RoboDK station: Coursework2_robot_manipulation.rdk

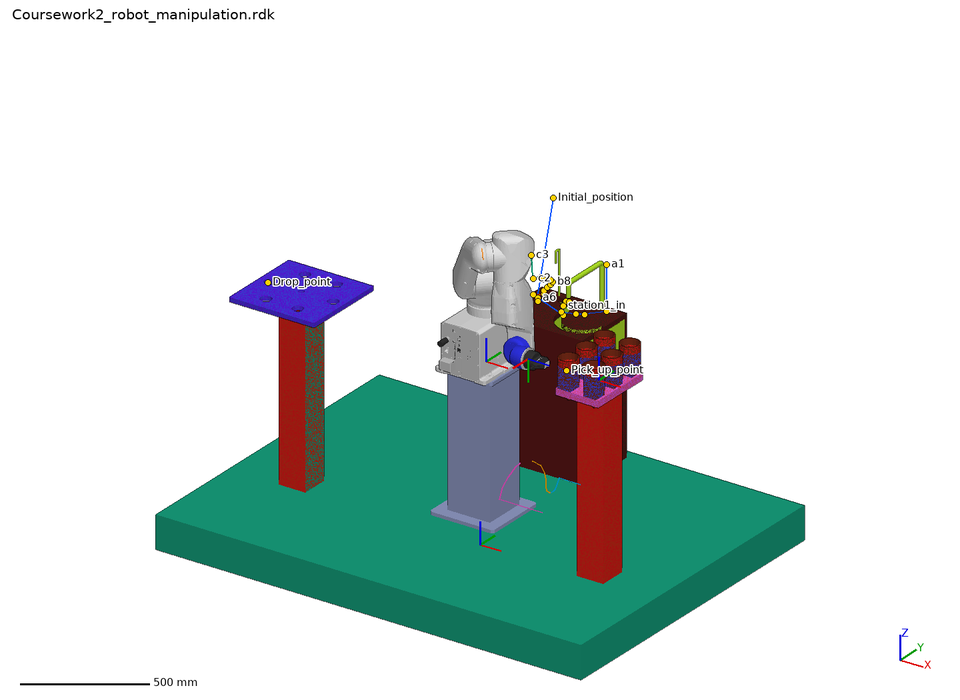
[picture v0: the station drawn from its stored meshes, robots at their saved joint values, targets as dots, program paths as lines]
Station Coursework2_robot_manipulator (saved by RoboDK 5.8.0). Poses are relative to the parent item; angles as X-Y-Z fixed-axis rotations.
Station parameters (name, value as stored): IO_5, 1
  - frame baseframe at (0, 0, 0) mm
    - object PDE4431_CW2_2024 at (0, 0, 0) mm, rotated rx 90 ry 0 rz 0 deg, size 2000 x 980 x 1500 mm, geometry from PDE4431_CW2_2024.STEP
    - frame Epson VT6 Base at (15, 20, 780) mm
      - robot Epson VT6: 6 axes, payload 6 kg, reach 920 mm, repeatability 0.1 mm, weight 40 kg
          modified DH rows (alpha deg, a mm, theta deg, d mm): 0, 0, 0, 412; -90, 100, -90, 0; 0, 420, 0, 0; -90, 0, 0, 400; 90, 0, 0, 0; -90, 0, 0, 80
          base shift (0, 0, 0) mm, rotated rx 0 ry 0 rz 90 deg
          joint limits [-170, -160, -51, -200, -125, -360] to [170, 65, 190, 200, 125, 360]; home [0, 0, 0, 0, 0, 0]; saved at [-133.764, -52.802, -29.005, -135.943, -84.093, 84.313]
        - tool Tool 1, TCP at (0, 0, 180) mm, rotated rx -90 ry 0 rz 0 deg
        - frame RobotiQ 2F-140 Gripper (Mechanism) Base at (0, 0, 0) mm
          - robot RobotiQ 2F-140 Gripper (Mechanism) (model RobotiQ 2F140): 1 axes, payload 5 kg
              joint limits [0] to [140]; home [140]; saved at [60]
    - frame input_area_reference_frame at (700, -200, 980) mm
      - object Cone-Part at (60, -120, 50) mm, rotated rx 90 ry 0 rz 90 deg, size 84.9 x 182 x 85 mm, geometry from Cone-Part.STEP
      - object Cone-Part at (60, 0, 50) mm, rotated rx 90 ry 0 rz 90 deg, size 84.9 x 182 x 85 mm, geometry from Cone-Part.STEP
      - object Cone-Part at (60, 120, 50) mm, rotated rx 90 ry 0 rz 90 deg, size 84.9 x 182 x 85 mm, geometry from Cone-Part.STEP
      - object Cone-Part at (-60, -120, 50) mm, rotated rx 90 ry 0 rz 90 deg, size 84.9 x 182 x 85 mm, geometry from Cone-Part.STEP
      - object Cone-Part at (-60, 0, 50) mm, rotated rx 90 ry 0 rz 90 deg, size 84.9 x 182 x 85 mm, geometry from Cone-Part.STEP
      - object Cone-Part at (-60, 120, 50) mm, rotated rx 90 ry 0 rz 90 deg, size 84.9 x 182 x 85 mm, geometry from Cone-Part.STEP
    - target Initial_position (Cartesian target) at (0, 493.22, 1288.03) mm, rotated rx 138 ry 0 rz 0 deg; joints [3.066, 29.719, -43.422, 4.791, -28.422, -96.269] of Epson VT6
    - target Gripper_open (Cartesian target) at (0.67, 380.04, 1461.97) mm, rotated rx -90 ry 0 rz 0 deg; joints [90, -0.57, 0.57, -89.99, -12.6, 0] of RobotiQ 2F-140 Gripper (Mechanism)
    - target Gripper_closed (Cartesian target) at (0.67, 380.04, 1461.97) mm, rotated rx -90 ry 0 rz 0 deg; joints [60, -0.57, 0.57, -89.99, -12.6, 0] of RobotiQ 2F-140 Gripper (Mechanism)
    - target Pick_up_point (Cartesian target) at (630, -320, 1050) mm, rotated rx 180 ry 0 rz -90 deg; joints [-121.329, -52.273, -41.785, -148.607, -93.465, 92.112] of Epson VT6
    - target station1_in (Cartesian target) at (107.17, 405.57, 892) mm, rotated rx 134.1 ry 22.52 rz 29.53 deg; joints [-42.76, -50.507, -48.896, -94.494, -48.491, -288.218] of Epson VT6
    - target station_in2 (Cartesian target) at (107.17, 425.58, 902) mm, rotated rx 154.09 ry 0 rz 49.53 deg; joints [-46.784, -59.524, -43.679, -90.222, -63.389, -255.291] of Epson VT6
    - target Station1_vert (Cartesian target) at (107.17, 445.58, 892) mm, rotated rx 180 ry 0 rz 49.53 deg; joints [-48.469, -79.022, -29.182, -82.396, -87.508, -251.961] of Epson VT6
    - target station1_return (Cartesian target) at (107.17, 405.57, 892) mm, rotated rx 134.1 ry 22.52 rz 29.53 deg; joints [-42.76, -50.507, -48.896, -94.494, -48.491, -288.218] of Epson VT6
    - target station1_retract2 (Cartesian target) at (107.17, 405.58, 852) mm, rotated rx 134.1 ry 22.52 rz 29.53 deg; joints [-42.76, -58.404, -45.922, -98.782, -49.061, -281.715] of Epson VT6
    - object Pedestal_4 at (14, 3, 150) mm, rotated rx 90 ry 0 rz 0 deg, size 300 x 630 x 300 mm, geometry from Pedestal_4.STEP
    - target Drop_point (Cartesian target) at (-765, -330, 1042) mm, rotated rx 180 ry 0 rz 90 deg; joints [124.2, -59.111, -6.959, -36.632, 70.399, -75.994] of Epson VT6
    - target a1 (Cartesian target) at (249.09, 493.26, 1072) mm, rotated rx 130 ry 0 rz 60.05 deg; joints [-44.186, -25.316, -23.381, -44.941, -61.89, 43.503] of Epson VT6
    - target a2 (Cartesian target) at (249.09, 493.26, 872) mm, rotated rx 130 ry 0 rz 60.05 deg; joints [-44.186, -51.38, -21.842, -59.131, -46.543, 67.327] of Epson VT6
    - target a3 (Cartesian target) at (194.9, 423.42, 872) mm, rotated rx 131.48 ry 11.84 rz 38.12 deg; joints [-47.351, -49.904, -38.58, -79.862, -43.086, 70.249] of Epson VT6
    - target a4 (Cartesian target) at (165.75, 406.79, 872) mm, rotated rx 134.36 ry 21.78 rz 37.08 deg; joints [-48.063, -53.054, -38.624, -75.536, -47.962, 62.433] of Epson VT6
    - target a5 (Cartesian target) at (109.56, 390.77, 872) mm, rotated rx 137.61 ry 29.5 rz 37.51 deg; joints [-45.93, -57.2, -41.919, -79.045, -51.807, 63.625] of Epson VT6
    - target a6 (Cartesian target) at (-2.03, 390.64, 902) mm, rotated rx 167.61 ry 29.5 rz 37.51 deg; joints [-40.605, -82.89, -49.926, -101.486, -85.95, 102.604] of Epson VT6
    - target b1 (Cartesian target) at (-13.32, 409.82, 877) mm, rotated rx 127 ry -33.83 rz -43.76 deg; joints [31.665, -52.224, -39.614, 69.659, -47.778, -224.233] of Epson VT6
    - target b2 (Cartesian target) at (-61.47, 446.95, 877) mm, rotated rx 120 ry 0 rz -61.45 deg; joints [27.592, -42.587, -43.484, 84.177, -30.167, -262.163] of Epson VT6
    - target b3 (Cartesian target) at (-30.23, 471.24, 877) mm, rotated rx 120 ry 0 rz -66.5 deg; joints [22.379, -42.928, -40.487, 79.841, -30.522, -256.952] of Epson VT6
    - target b4 (Cartesian target) at (-44.93, 495.72, 877) mm, rotated rx 120 ry 0 rz -75.12 deg; joints [22.759, -44.277, -33.238, 62.836, -33.826, -247.376] of Epson VT6
    - target b6 (Cartesian target) at (-53.08, 528.17, 877) mm, rotated rx 120 ry 0 rz -85.53 deg; joints [21.649, -46.651, -24.32, 48.543, -39.597, -240.743] of Epson VT6
    - target b7 (Cartesian target) at (-54.53, 553.97, 877) mm, rotated rx 120 ry 0 rz -103.24 deg; joints [19.178, -50.022, -14.03, 34.25, -48.589, -240.495] of Epson VT6
    - target b8 (Cartesian target) at (-65.31, 579.52, 877) mm, rotated rx 120 ry 0 rz -35.21 deg; joints [18.907, -44.258, -33.32, 103.859, -24.661, -245.312] of Epson VT6
    - target b9 (Cartesian target) at (-81.16, 591.33, 877) mm, rotated rx 120 ry 0 rz -15.6 deg; joints [16.379, -43.789, -35.498, 133.999, -21.601, -254.488] of Epson VT6
    - target b10 (Cartesian target) at (-105.52, 575.28, 877) mm, rotated rx 120 ry 0 rz -5.76 deg; joints [17.409, -43.261, -38.323, 149.049, -22.485, -261.342] of Epson VT6
    - target c1 (Cartesian target) at (-126.7, 587.41, 877) mm, rotated rx 121.57 ry -17.23 rz 40.16 deg; joints [13.883, -45.369, -39.632, 180.61, -30.533, -239.449] of Epson VT6
    - target c2 (Cartesian target) at (-143.48, 560.98, 877) mm, rotated rx 121.57 ry -17.23 rz 52.76 deg; joints [12.465, -9.414, 61.191, 171.217, 106.936, -230.002] of Epson VT6
    - target c3 (Cartesian target) at (-146.17, 555.68, 977) mm, rotated rx 127 ry -33.83 rz 40.31 deg; joints [23.435, -32.385, -50.82, 158.038, -42.083, -218.54] of Epson VT6
  - Python program Full1_program (listed below)
  - program Gripper_Open (2 instructions, listed below)
  - program Gripper_close (1 instructions, listed below)
  - program Gripper_fn_detach (1 instructions, listed below)
  - program Gripper_fn_attach (1 instructions, listed below)
  - program Arc1 (15 instructions, listed below)
  - Python program arc1_repeat (listed below)
  - program Arc2 (12 instructions, listed below)
  - Python program arc2_repeat (listed below)
  - program Arc3 (5 instructions, listed below)
  - program Reset_prog (1 instructions, listed below)
  - object Curve1 at (0, 0, 832) mm, geometry from Imported curve
  - machining project Path1 settings: rotZ(0) | rotX(0)*rotY(0) | onStart | onPathStart | onApproach | onPoint | onRetract | onFinish | SetRPM(%1) | SetTool(%1) | Extruder(%1) | default | default | OutOnMov(%1) | OutOffMov(%1) | onPathFinish | M_RunCode(%1)
  - program Path1 (17 instructions, listed below)
  - object Curve2 at (0, 0, 832) mm, geometry from 000000
  - machining project Path2 settings: rotZ(0) | rotX(0)*rotY(0) | onStart | onPathStart | onApproach | onPoint | onRetract | onFinish | SetRPM(%1) | SetTool(%1) | Extruder(%1) | default | default | OutOnMov(%1) | OutOffMov(%1) | onPathFinish | M_RunCode(%1)
  - program Path2 (24 instructions, listed below)
  - object Curve3 at (0, 0, 832) mm
  - machining project Path3 settings: rotZ(0) | rotX(0)*rotY(0) | onStart | onPathStart | onApproach | onPoint | onRetract | onFinish | SetRPM(%1) | SetTool(%1) | Extruder(%1) | default | default | OutOnMov(%1) | OutOffMov(%1) | onPathFinish | M_RunCode(%1)
  - program Path3 (17 instructions, listed below)
  - Python program pick (listed below)
  - Python program drop (listed below)
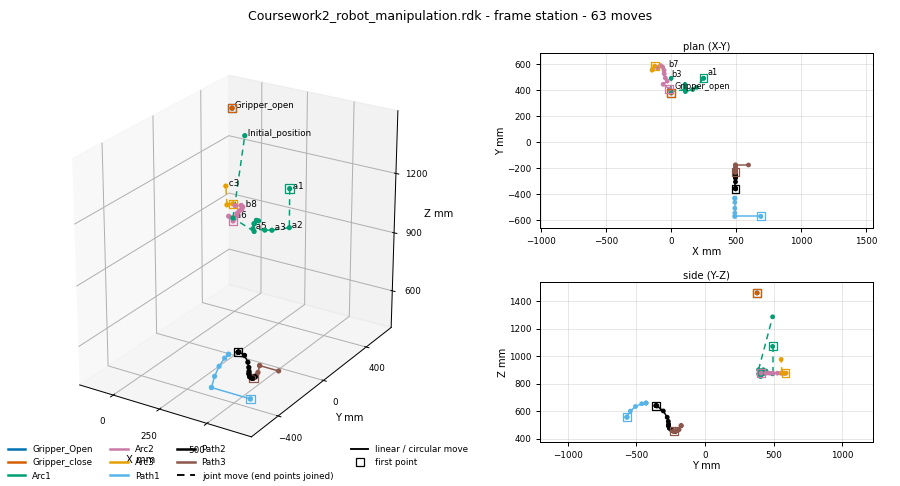
[picture p0: tool path of Coursework2_robot_manipulation.rdk in frame station, 63 of 63 moves have a stored position in this frame; points joined in program order, loops and branches not executed]

--- Python program Full1_program ---
from robodk.robolink import *
from robodk.robomath import *
import time

#Connection b/w roboDK
RDK=Robolink()

#conf. robot
robot=RDK.Item('Epson VT6')

robot.setSpeed(100)

base = RDK.Item('baseframe')
end_effector =RDK.Item('RobotiQ 2F-140 Gripper (Mechanism) Base')

#setting home position
home = RDK.Item('Initial_position')

#Pick_up_points with one point reference
pickup1=RDK.Item('Pick_up_point')
pickup2=pickup1.Pose()*transl(-120,0,0)
pickup3=pickup1.Pose()*transl(-240,0,0)
pickup4=pickup1.Pose()*transl(0,-120,0)
pickup5=pickup1.Pose()*transl(-120,-120,0)
pickup6=pickup1.Pose()*transl(-240,-120,0)

pickup=[pickup3,pickup2,pickup1,pickup6,pickup5,pickup4]

#pickup_approach
pa1=pickup1.Pose()*transl(0,0,-80)
pa2=pickup1.Pose()*transl(-120,0,-80)
pa3=pickup1.Pose()*transl(-240,0,-80)
pa4=pickup1.Pose()*transl(0,-120,-80)
pa5=pickup1.Pose()*transl(-120,-120,-80)
pa6=pickup1.Pose()*transl(-240,-120,-80)

pa7=pickup1.Pose()*transl(-300,-20,-80)

pa=[pa3,pa2,pa1,pa6,pa5,pa4]

#Drop_points with one point reference
drop1=RDK.Item('Drop_point')
drop2=drop1.Pose()*transl(129.9,-75,0)
drop3=drop1.Pose()*transl(259.8,0,0)
drop4=drop1.Pose()*transl(0,150,0)
drop5=drop1.Pose()*transl(129.9,225,0)
drop6=drop1.Pose()*transl(259.8,150,0)



drop=[drop1,drop2,drop3,drop4,drop5,drop6]

#drop_approach
da1=drop1.Pose()*transl(0,0,-80)
da2=drop1.Pose()*transl(129.9,-75,-80)
da3=drop1.Pose()*transl(259.8,0,-80)
da4=drop1.Pose()*transl(0,150,-80)
da5=drop1.Pose()*transl(129.9,225,-80)
da6=drop1.Pose()*transl(259.8,150,-80)

da7=drop1.Pose()*transl(320,150,-80)
da8=drop1.Pose()*transl(129,75,-80)
da=[da1,da2,da3,da4,da5,da6]

#Call_functions
grip_on=RDK.Item('Gripper_close')
grip_off=RDK.Item('Gripper_Open')
attach=RDK.Item('Gripper_fn_attach')
detach=RDK.Item('Gripper_fn_detach')

#arc_functions
Station1_curve=RDK.Item('Curve')
Station2_curve=RDK.Item('Curve2')

#station1_filling_area targets for station 1
s1_in1=RDK.Item('station1_in')
s1_in2=RDK.Item('station_in2')
s1_vert=RDK.Item('Station1_vert')
s1_out1=RDK.Item('station1_return')
s1_out2=RDK.Item('station1_retract2')

#reset function
reset=RDK.Item('Reset_prog')

def arc_1():

    #setting home position
    home = RDK.Item('Initial_position')

    #station1_filling_area targets for curve
    arc_approach=RDK.Item('a1')
    curve_start=RDK.Item('a2')
    curve_start1=curve_start.Pose()*transl(0,0,1)
    curve_center1=RDK.Item('a3')
    curve_center2=RDK.Item('a4')
    curve_end=RDK.Item('a5')
    curve_exit=RDK.Item('a6')

    #station1_filling_area targets for station 1
    s1_in1=RDK.Item('station1_in')
    s1_in2=RDK.Item('station_in2')
    s1_vert=RDK.Item('Station1_vert')
    s1_out1=RDK.Item('station1_return')
    s1_out2=RDK.Item('station1_retract2')

    #curve movement
    robot.MoveJ(arc_approach)
    robot.MoveL(curve_start)
    robot.MoveC(curve_start1,curve_center1)
    robot.MoveC(curve_center2,curve_end)

    #filling function
    robot.MoveL(s1_in1)
    robot.MoveL(s1_in2)
    robot.MoveL(s1_vert)
    pause(1)
    for i in range(3):
        increment=i*2
        robot.MoveL(s1_vert.Pose()*transl(-18,18,increment))
        robot.MoveL(s1_vert.Pose()*transl(18,18,increment))
        robot.MoveL(s1_vert.Pose()*transl(18,-18,increment))
        robot.MoveL(s1_vert.Pose()*transl(-18,-18,increment))
        robot.MoveL(s1_vert.Pose()*transl(-18,18,increment))
    robot.MoveL(s1_out1)
    robot.MoveL(s1_out2)
    robot.MoveL(curve_exit)
    robot.MoveJ(home)

def arc_2():

    #setting home position
    home = RDK.Item('Initial_position')

    #station1_filling_area targets for curve
    arc_approach=RDK.Item('b1')
    p1=RDK.Item('b2')
    p2=RDK.Item('b3')
    p3=RDK.Item('b4')
    p4=RDK.Item('b5')
    p5=RDK.Item('b6')
    p6=RDK.Item('b7')
    p7=RDK.Item('b8')
    p8=RDK.Item('b9')
    p9=RDK.Item('b10')


    #curve movement
    robot.MoveJ(arc_approach)

    robot.MoveL(p1)
    robot.MoveL(p2)
    robot.MoveL(p3)

    robot.MoveL(p5)
    robot.MoveL(p6)
    robot.MoveL(p7)
    robot.MoveL(p8)
    robot.MoveL(p9)
    pause(.5)
    for i in range(3):
        increment=i*5
        robot.MoveL(p9.Pose()*transl(-18,18,increment))
        robot.MoveL(p9.Pose()*transl(18,18,increment))
        robot.MoveL(p9.Pose()*transl(18,-18,increment))
        robot.MoveL(p9.Pose()*transl(-18,-18,increment))
        robot.MoveL(p9.Pose()*transl(-18,18,increment))


def arc_3():

    p1=RDK.Item('c1')
    p2=RDK.Item('c2')
    p3=RDK.Item('c3')

    robot.MoveL(p1)
    robot.MoveL(p2)
    robot.MoveL(p3)

reset.RunProgram()
robot.MoveJ(home)

for i in range(6):

    robot.MoveJ(home)

    approach=pa[i]
    robot.MoveJ(approach)

    pick_position=pickup[i]
    robot.MoveL(pick_position)

    grip_on.RunProgram()
    attach.RunProgram()


    robot.MoveL(approach)
    robot.MoveL(pa7)

    arc_1()
    arc_2()
    arc_3()


    robot.MoveJ(da7)
    robot.MoveL(da6)
    drop_approach=da[i]
    robot.MoveL(drop_approach)

    drop_position=drop[i]
    robot.MoveL(drop_position)

    grip_off.RunProgram()
    detach.RunProgram()

    pause(1)

    robot.MoveL(drop_approach)

robot.MoveJ(home)

--- program Gripper_Open (robot RobotiQ 2F-140 Gripper (Mechanism)) ---
  MoveJ (Gripper_open)
  Pause 2.0 s

--- program Gripper_close (robot RobotiQ 2F-140 Gripper (Mechanism)) ---
  MoveJ (Gripper_closed)

--- program Gripper_fn_detach (robot Epson VT6) ---
  Detach from Tool 1

--- program Gripper_fn_attach (robot Epson VT6) ---
  Attach to Tool 1

--- program Arc1 (robot Epson VT6) ---
  Set Ref.: baseframe
  Set Tool: Tool 1
  MoveJ (a1)
  MoveJ (a2)
  MoveJ (a3)
  MoveJ (a4)
  MoveJ (a5)
  MoveL (station1_in)
  MoveL (station_in2)
  MoveL (Station1_vert)
  Pause 500 ms
  MoveL (station1_return)
  MoveL (station1_retract2)
  MoveJ (a6)
  MoveJ (Initial_position)

--- Python program arc1_repeat ---
from robodk.robolink import *
from robodk.robomath import *
import time

#Connection b/w roboDK
RDK=Robolink()

#conf. robot
robot=RDK.Item('Epson VT6')

def repeat():

    s1_vert=RDK.Item('Station1_vert')
    for i in range(3):
        increment=i*2
        robot.MoveL(s1_vert.Pose()*transl(-18,18,increment))
        robot.MoveL(s1_vert.Pose()*transl(18,18,increment))
        robot.MoveL(s1_vert.Pose()*transl(18,-18,increment))
        robot.MoveL(s1_vert.Pose()*transl(-18,-18,increment))
        robot.MoveL(s1_vert.Pose()*transl(-18,18,increment))
repeat()

--- program Arc2 (robot Epson VT6) ---
  Set Ref.: baseframe
  Set Tool: Tool 1
  MoveJ (b1)
  MoveL (b2)
  MoveL (b3)
  MoveL (b4)
  MoveL (b6)
  MoveL (b7)
  MoveL (b8)
  MoveL (b9)
  MoveL (b10)
  Call arc2_repeat

--- Python program arc2_repeat ---
from robodk.robolink import *
from robodk.robomath import *
import time

#Connection b/w roboDK
RDK=Robolink()

#conf. robot
robot=RDK.Item('Epson VT6')

def repeat():

    p9=RDK.Item('b10')
    for i in range(3):
        increment=i*5
        robot.MoveJ(p9.Pose()*transl(-18,18,increment))
        robot.MoveJ(p9.Pose()*transl(18,18,increment))
        robot.MoveJ(p9.Pose()*transl(18,-18,increment))
        robot.MoveJ(p9.Pose()*transl(-18,-18,increment))
        robot.MoveJ(p9.Pose()*transl(-18,18,increment))
repeat()

--- program Arc3 (robot Epson VT6) ---
  Set Ref.: baseframe
  Set Tool: Tool 1
  MoveJ (c1)
  MoveJ (c2)
  MoveJ (c3)

--- program Reset_prog (robot Epson VT6) ---
  Replace objects

--- program Path1 (robot Epson VT6) ---
  Smooth(1)
  Set speed (1000.0 mm/s)
  Set Ref.: RobotiQ 2F-140 Gripper (Mechanism) Base
  Set Tool: Tool 1
  Show Tool 1
  MoveJ 1 to (249.09, 493.26, 240) mm, rotated rx 130 ry 0 rz 60.05 deg; joints [-44.186, -25.316, -23.381, -44.941, -61.89, 43.503]
  MoveL 2 to (249.09, 493.26, 240) mm, rotated rx 130 ry 0 rz 60.05 deg; joints [-44.186, -25.316, -23.381, -44.941, -61.89, 43.503]
  MoveL 3 to (249.09, 493.26, 40) mm, rotated rx 130 ry 0 rz 60.05 deg; joints [-44.186, -51.38, -21.842, -59.131, -46.543, 67.327]
  MoveL 4 to (249.09, 493.26, 40) mm, rotated rx 130 ry 0 rz 60.05 deg; joints [-44.186, -51.38, -21.842, -59.131, -46.543, 67.327]
  Set speed (50.0 mm/s)
  MoveL 5 to (223.76, 449.31, 40) mm, rotated rx 130 ry 0 rz 41.9 deg; joints [-46.416, -48.516, -37.52, -86.959, -40.047, 83.835]
  MoveL 6 to (186.76, 416.11, 40) mm, rotated rx 131.76 ry 15.19 rz 37.08 deg; joints [-47.66, -50.503, -38.869, -78.271, -44.082, 66.939]
  MoveL 7 to (141.07, 395.85, 40) mm, rotated rx 137.61 ry 29.5 rz 37.51 deg; joints [-48.444, -56.619, -38.327, -73.341, -52.504, 58.401]
  MoveL 8 to (109.56, 390.77, 40) mm, rotated rx 137.61 ry 29.5 rz 37.51 deg; joints [-45.93, -57.2, -41.919, -79.045, -51.807, 63.625]
  Set speed (1000.0 mm/s)
  MoveL 9 to (109.56, 390.77, 40) mm, rotated rx 137.61 ry 29.5 rz 37.51 deg; joints [-45.93, -57.2, -41.919, -79.045, -51.807, 63.625]
  MoveL 10 to (109.56, 390.77, 40) mm, rotated rx 137.61 ry 29.5 rz 37.51 deg; joints [-45.93, -57.2, -41.919, -79.045, -51.807, 63.625]

--- program Path2 (robot Epson VT6) ---
  Smooth(1)
  Set speed (1000.0 mm/s)
  Set Ref.: RobotiQ 2F-140 Gripper (Mechanism) Base
  Set Tool: Tool 1
  Show Tool 1
  MoveJ 1 to (36.68, 409.82, 45) mm, rotated rx 127 ry -33.83 rz -43.76 deg; joints [25.483, -52.5, -42.953, 79.119, -47.184, -229.095]
  MoveL 2 to (36.68, 409.82, 45) mm, rotated rx 127 ry -33.83 rz -43.76 deg; joints [25.483, -52.5, -42.953, 79.119, -47.184, -229.095]
  MoveL 3 to (36.68, 409.82, 45) mm, rotated rx 127 ry -33.83 rz -43.76 deg; joints [25.483, -52.5, -42.953, 79.119, -47.184, -229.095]
  MoveL 4 to (36.68, 409.82, 45) mm, rotated rx 127 ry -33.83 rz -43.76 deg; joints [25.483, -52.5, -42.953, 79.119, -47.184, -229.095]
  Set speed (50.0 mm/s)
  MoveL 5 to (30.33, 412.26, 45) mm, rotated rx 121.57 ry -17.23 rz -48.2 deg; joints [20.334, -45.22, -48.276, 90.637, -35.42, -245.38]
  MoveL 6 to (-16.31, 448.54, 45) mm, rotated rx 120 ry 0 rz -58.48 deg; joints [21.513, -42.402, -46.974, 98.943, -29.897, -268.767]
  MoveL 7 to (-44.67, 494.77, 45) mm, rotated rx 120 ry 0 rz -74.82 deg; joints [22.785, -44.219, -33.495, 63.332, -33.683, -247.647]
  MoveL 8 to (-52.69, 524.33, 45) mm, rotated rx 120 ry 0 rz -84.24 deg; joints [21.854, -46.338, -25.378, 49.984, -38.848, -241.279]
  MoveL 9 to (-54.72, 544.48, 45) mm, rotated rx 120 ry 0 rz -91 deg; joints [20.763, -48.074, -19.769, 42.981, -42.932, -239.054]
  MoveL 10 to (-54.56, 553.85, 45) mm, rotated rx 120 ry 0 rz -104.22 deg; joints [19.069, -50.132, -13.72, 33.645, -48.97, -240.77]
  MoveL 11 to (-53.46, 558.18, 45) mm, rotated rx 120 ry 0 rz -68.78 deg; joints [21.114, -46.203, -25.842, 61.98, -34.499, -237.024]
  MoveL 12 to (-60.04, 575.11, 45) mm, rotated rx 120 ry 0 rz -39.91 deg; joints [19.184, -44.365, -32.855, 97.818, -25.659, -244.004]
  MoveL 13 to (-77.38, 589.61, 45) mm, rotated rx 120 ry 0 rz -24.46 deg; joints [17.953, -44.094, -34.057, 118.542, -22.577, -248.854]
  MoveL 14 to (-85.36, 593.25, 45) mm, rotated rx 120 ry 0 rz -5.76 deg; joints [14.331, -43.583, -36.541, 151.333, -20.975, -260.528]
  MoveL 15 to (-105.52, 595.28, 45) mm, rotated rx 120 ry 0 rz -5.76 deg; joints [16.673, -43.805, -35.421, 146.854, -20.42, -258.204]
  Set speed (1000.0 mm/s)
  MoveL 16 to (-105.52, 595.28, 45) mm, rotated rx 120 ry 0 rz -5.76 deg; joints [16.673, -43.805, -35.421, 146.854, -20.42, -258.204]
  MoveL 17 to (-105.52, 595.28, 45) mm, rotated rx 120 ry 0 rz -5.76 deg; joints [16.673, -43.805, -35.421, 146.854, -20.42, -258.204]

--- program Path3 (robot Epson VT6) ---
  Smooth(1)
  Set speed (1000.0 mm/s)
  Set Ref.: RobotiQ 2F-140 Gripper (Mechanism) Base
  Set Tool: Tool 1
  Show Tool 1
  MoveJ 1 to (-91.28, 595.7, 45) mm, rotated rx 120 ry 0 rz -1.36 deg; joints [13.786, -43.606, -36.42, 158.126, -20.523, -262.585]
  MoveL 2 to (-91.28, 595.7, 45) mm, rotated rx 120 ry 0 rz -1.36 deg; joints [13.786, -43.606, -36.42, 158.126, -20.523, -262.585]
  MoveL 3 to (-91.28, 595.7, 45) mm, rotated rx 120 ry 0 rz -1.36 deg; joints [13.786, -43.606, -36.42, 158.126, -20.523, -262.585]
  MoveL 4 to (-91.28, 595.7, 45) mm, rotated rx 120 ry 0 rz -1.36 deg; joints [13.786, -43.606, -36.42, 158.126, -20.523, -262.585]
  Set speed (50.0 mm/s)
  MoveL 5 to (-106.2, 596.05, 45) mm, rotated rx 120 ry 0 rz 16.66 deg; joints [10.53, -43.615, -36.376, 188.951, -20.074, -273.101]
  MoveL 6 to (-120.02, 591.91, 45) mm, rotated rx 121.57 ry -17.23 rz 23.67 deg; joints [18.455, -45.541, -38.15, 155.717, -29.695, -234.898]
  MoveL 7 to (-131.8, 583.97, 45) mm, rotated rx 121.57 ry -17.23 rz 52.76 deg; joints [10.316, -45.412, -39.236, 199.254, -30.439, -242.392]
  MoveL 8 to (-146.17, 555.68, 45) mm, rotated rx 121.57 ry -17.23 rz 52.76 deg; joints [12.99, -45.124, -42.873, 194.754, -33.591, -240.235]
  Set speed (1000.0 mm/s)
  MoveL 9 to (-146.17, 555.68, 45) mm, rotated rx 121.57 ry -17.23 rz 52.76 deg; joints [12.99, -45.124, -42.873, 194.754, -33.591, -240.235]
  MoveL 10 to (-146.17, 555.68, 145) mm, rotated rx 127 ry -33.83 rz 40.31 deg; joints [23.435, -32.385, -50.82, 158.038, -42.083, -218.54]

--- Python program pick ---
from robodk.robolink import *
from robodk.robomath import *
import time

#Connection b/w roboDK
RDK=Robolink()

#conf. robot
robot=RDK.Item('Epson VT6')

robot.setSpeed(100)

base = RDK.Item('baseframe')
end_effector =RDK.Item('RobotiQ 2F-140 Gripper (Mechanism) Base')

#setting home position
home = RDK.Item('Initial_position')

#Pick_up_points with one point reference
pickup1=RDK.Item('Pick_up_point')
pickup2=pickup1.Pose()*transl(-120,0,0)
pickup3=pickup1.Pose()*transl(-240,0,0)
pickup4=pickup1.Pose()*transl(0,-120,0)
pickup5=pickup1.Pose()*transl(-120,-120,0)
pickup6=pickup1.Pose()*transl(-240,-120,0)

pickup=[pickup3,pickup2,pickup1,pickup6,pickup5,pickup4]

#pickup_approach
pa1=pickup1.Pose()*transl(0,0,-80)
pa2=pickup1.Pose()*transl(-120,0,-80)
pa3=pickup1.Pose()*transl(-240,0,-80)
pa4=pickup1.Pose()*transl(0,-120,-80)
pa5=pickup1.Pose()*transl(-120,-120,-80)
pa6=pickup1.Pose()*transl(-240,-120,-80)

pa7=pickup1.Pose()*transl(-300,-20,-80)

pa=[pa3,pa2,pa1,pa6,pa5,pa4]

#Drop_points with one point reference
drop1=RDK.Item('Drop_point')
drop2=drop1.Pose()*transl(129.9,-75,0)
drop3=drop1.Pose()*transl(259.8,0,0)
drop4=drop1.Pose()*transl(0,150,0)
drop5=drop1.Pose()*transl(129.9,225,0)
drop6=drop1.Pose()*transl(259.8,150,0)



drop=[drop1,drop2,drop3,drop4,drop5,drop6]

#drop_approach
da1=drop1.Pose()*transl(0,0,-80)
da2=drop1.Pose()*transl(129.9,-75,-80)
da3=drop1.Pose()*transl(259.8,0,-80)
da4=drop1.Pose()*transl(0,150,-80)
da5=drop1.Pose()*transl(129.9,225,-80)
da6=drop1.Pose()*transl(259.8,150,-80)

da7=drop1.Pose()*transl(320,150,-80)
da8=drop1.Pose()*transl(129,75,-80)
da=[da1,da2,da3,da4,da5,da6]


robot.MoveJ(home)

robot.MoveJ(pa3)

robot.MoveL(pickup3)

robot.MoveL(pa3)
robot.MoveJ(pa7)


"""
    robot.MoveJ(da7)
    robot.MoveL(da6)

    drop_approach=da[i]
    robot.MoveL(drop_approach)

    drop_position=drop[i]
    robot.MoveL(drop_position)


    pause(1)

    robot.MoveL(drop_approach)

robot.MoveJ(home)
"""

--- Python program drop ---
from robodk.robolink import *
from robodk.robomath import *
import time

#Connection b/w roboDK
RDK=Robolink()

#conf. robot
robot=RDK.Item('Epson VT6')

robot.setSpeed(100)

base = RDK.Item('baseframe')
end_effector =RDK.Item('RobotiQ 2F-140 Gripper (Mechanism) Base')

#setting home position
home = RDK.Item('Initial_position')

#Pick_up_points with one point reference
pickup1=RDK.Item('Pick_up_point')
pickup2=pickup1.Pose()*transl(-120,0,0)
pickup3=pickup1.Pose()*transl(-240,0,0)
pickup4=pickup1.Pose()*transl(0,-120,0)
pickup5=pickup1.Pose()*transl(-120,-120,0)
pickup6=pickup1.Pose()*transl(-240,-120,0)

pickup=[pickup3,pickup2,pickup1,pickup6,pickup5,pickup4]

#pickup_approach
pa1=pickup1.Pose()*transl(0,0,-80)
pa2=pickup1.Pose()*transl(-120,0,-80)
pa3=pickup1.Pose()*transl(-240,0,-80)
pa4=pickup1.Pose()*transl(0,-120,-80)
pa5=pickup1.Pose()*transl(-120,-120,-80)
pa6=pickup1.Pose()*transl(-240,-120,-80)

pa7=pickup1.Pose()*transl(-300,-20,-80)

pa=[pa3,pa2,pa1,pa6,pa5,pa4]

#Drop_points with one point reference
drop1=RDK.Item('Drop_point')
drop2=drop1.Pose()*transl(129.9,-75,0)
drop3=drop1.Pose()*transl(259.8,0,0)
drop4=drop1.Pose()*transl(0,150,0)
drop5=drop1.Pose()*transl(129.9,225,0)
drop6=drop1.Pose()*transl(259.8,150,0)



drop=[drop1,drop2,drop3,drop4,drop5,drop6]

#drop_approach
da1=drop1.Pose()*transl(0,0,-80)
da2=drop1.Pose()*transl(129.9,-75,-80)
da3=drop1.Pose()*transl(259.8,0,-80)
da4=drop1.Pose()*transl(0,150,-80)
da5=drop1.Pose()*transl(129.9,225,-80)
da6=drop1.Pose()*transl(259.8,150,-80)

da7=drop1.Pose()*transl(320,150,-80)
da8=drop1.Pose()*transl(129,75,-80)
da=[da1,da2,da3,da4,da5,da6]


robot.MoveJ(da7)
robot.MoveL(da6)

robot.MoveJ(da1)

robot.MoveL(drop1)

robot.MoveJ(da1)

robot.MoveJ(home)
